TYPE (* One term of one interlock alternative. TermCount>=1 heads an alternative and counts its terms; 0 continues the one above. *)
  (* Standard: 1131-3 *)
  (* Version 0.1, 5/24/2026, easensoy, WMG, array-of-struct packaging of the 4 Rule arrays *)
  PACKAGE Main;
  InterlockRule : STRUCT
    FromState : INT;
    ToState : INT;
    SourceID : INT;
    BlockedState : INT;
    TermCount : INT;
  END_STRUCT;
END_TYPE
